(* CoDeSys 2.3 export: PLC_PRG_.EXP *)

(* POU PLC_PRG_, FBD *)
PROGRAM PLC_PRG_
VAR
	PWM_husillo: PWM;
	PID_husillo: PID;
	sp_husillo: REAL;
	salida_husillo: REAL;
	ENABLE: BOOL;
	salida_husillo_int: INT;
	TN_h: REAL:=0.08;
	TV_h: REAL:=0.08;
	KP_h: REAL:=0.1;
	TN_n: REAL:=0.08;
	TV_n: REAL:=0.08;
	KP_n: REAL:=0.1;
	PWM_nozzle: PWM;
	salida_nozzle: REAL;
	salida_nozzle_int: INT;
	PID_nozzle: PID;
	sp_nozzle: REAL;
	PID_RESET_h: BOOL;
	PID_RESET_n: BOOL;
	OVERFLOW_h: BOOL;
	OVERFLOW_n: BOOL;
	lim_h: BOOL;
	Volt_diametro: REAL;
	Diametro_mm: REAL;
	SD_WRITE: SD_WRITE;
	DIM: DWORD;
	dim_word: DWORD;
	diametro_puntero: DWORD;
	DONE: BOOL;
	ERR: BOOL;
	ERNO: WORD;
	SD_ENABLE: BOOL;
	kk: R_TRIG;
	SEG: DWORD;
	FILENO: BYTE:=0;
	Diametro_string: STRING;
	datos: STRING;
	FILE_Write: FILE_Write;
	FILE_Open: FILE_Open;
	hfile: CAA_HANDLE;
	fileName: STRING(80) :=  'sdcard/plan.csv';
	FileMode				: FILE_MODE		:= FILE_MAPPD;
	FILE_Close: FILE_Close;
	CLOCK: CLOCK;
	hora: DWORD;
	eError: FILE_ERROR;
	Escritura: Write_SD_Card;
	SR_enable: SR;
END_VAR
VAR CONSTANT
	CRLF: STRING := '$r$n';					(* New line *)
	SEMIKOLON : STRING(1) :=';';
END_VAR
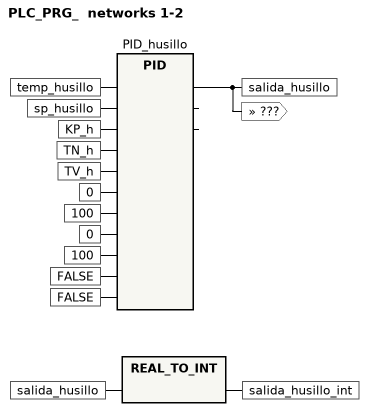
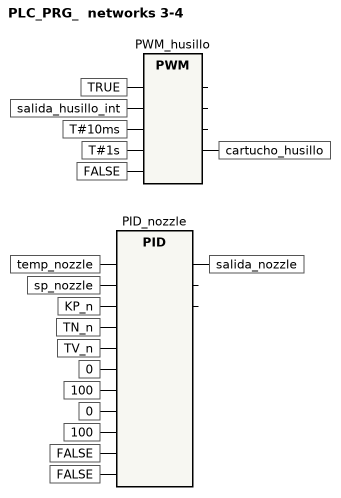
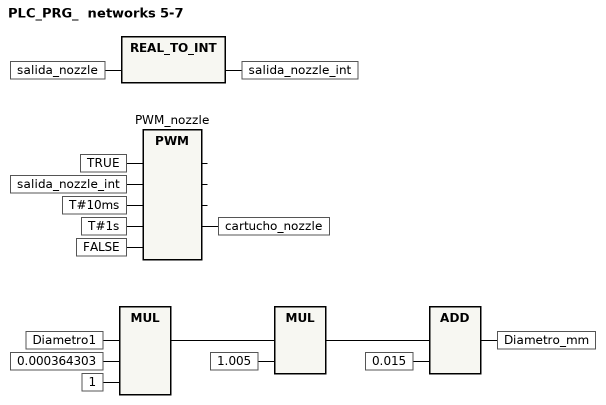
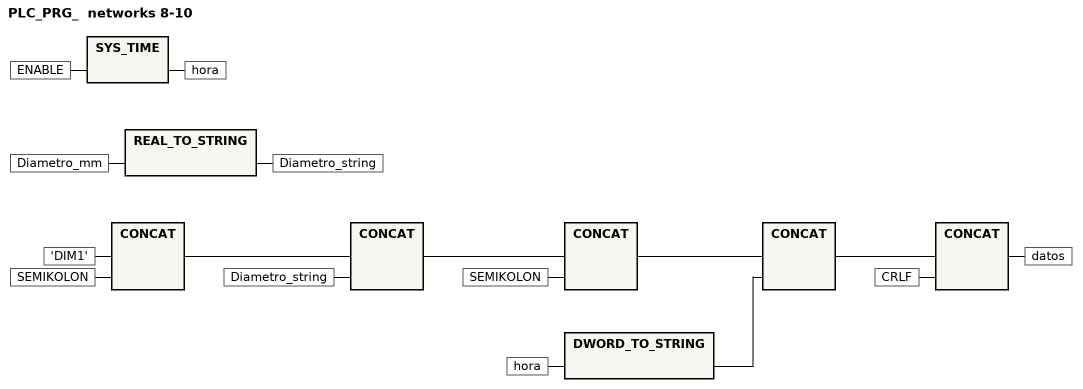
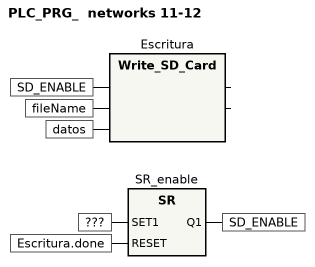
_FBD_ (* Function Block Diagram *)
NETWORK 1
	<PID_husillo:PID(temp_husillo, sp_husillo, KP_h, TN_h, TV_h, 0, 100, 0, 100, FALSE, FALSE) => salida_husillo> => >>???
NETWORK 2
	REAL_TO_INT(salida_husillo) => salida_husillo_int
NETWORK 3
	PWM_husillo:PWM(TRUE, salida_husillo_int, T#10ms, T#1s, FALSE, out 4 => cartucho_husillo)
NETWORK 4
	PID_nozzle:PID(temp_nozzle, sp_nozzle, KP_n, TN_n, TV_n, 0, 100, 0, 100, FALSE, FALSE) => salida_nozzle
NETWORK 5
	REAL_TO_INT(salida_nozzle) => salida_nozzle_int
NETWORK 6
	PWM_nozzle:PWM(TRUE, salida_nozzle_int, T#10ms, T#1s, FALSE, out 4 => cartucho_nozzle)
NETWORK 7
	ADD(MUL(MUL(Diametro1, 0.000364303, 1), 1.005), 0.015) => Diametro_mm
NETWORK 8
	SYS_TIME(ENABLE) => hora
NETWORK 9
	REAL_TO_STRING(Diametro_mm) => Diametro_string
NETWORK 10
	CONCAT(CONCAT(CONCAT(CONCAT(CONCAT('DIM1', SEMIKOLON), Diametro_string), SEMIKOLON), DWORD_TO_STRING(hora)), CRLF) => datos
NETWORK 11
	Escritura:Write_SD_Card(SD_ENABLE, fileName, datos)
NETWORK 12
	SR_enable:SR(SET1: ???, RESET: Escritura.done) => SD_ENABLE
_END_FBD_
END_PROGRAM
